// TIA Portal V17 export
// export: Created 2024-08-26T21:10:50.1762812Z, ExportSetting WithDefaults, DisplayName Totally Integrated Automation Portal, DisplayVersion V17 Update 7, DisplayName TIA Portal Openness, DisplayVersion V17 Update 7, DisplayName TIA Portal Version Control Interface, DisplayVersion V17, DisplayName SINAMICS Startdrive Advanced, DisplayVersion V17 SP2, DisplayName SINAMICS Startdrive G110M, G120, G120C, G120D, G120P, G115D, DisplayVersion V17 SP2, DisplayName SINAMICS Startdrive G130, G150, S120, S150, SINAMICS MV, S210, DisplayVersion V17 SP2, DisplayName STEP 7 Professional, DisplayVersion V17 Update 7, DisplayName STEP 7 Safety, DisplayVersion V17 Update 6, DisplayName WinCC Advanced / Unified PC, DisplayVersion V17 Update 7
FUNCTION "stationAlarms" : Void   // FC2, LAD
{ S7_Optimized_Access := 'TRUE' }
VERSION : 0.1
// stored: AutoNumber true, IsIECCheckEnabled false, SetENOAutomatically false, UDAEnableTagReadback false
   VAR_TEMP   // added for the SCL form of the ladder/FBD networks
      _w1 : Bool;
      _w2 : Bool;
      _w3 : Bool;
      _w4 : Bool;
      _w5 : Bool;
   END_VAR
BEGIN

REGION Network 1: ACTIVE ALARM
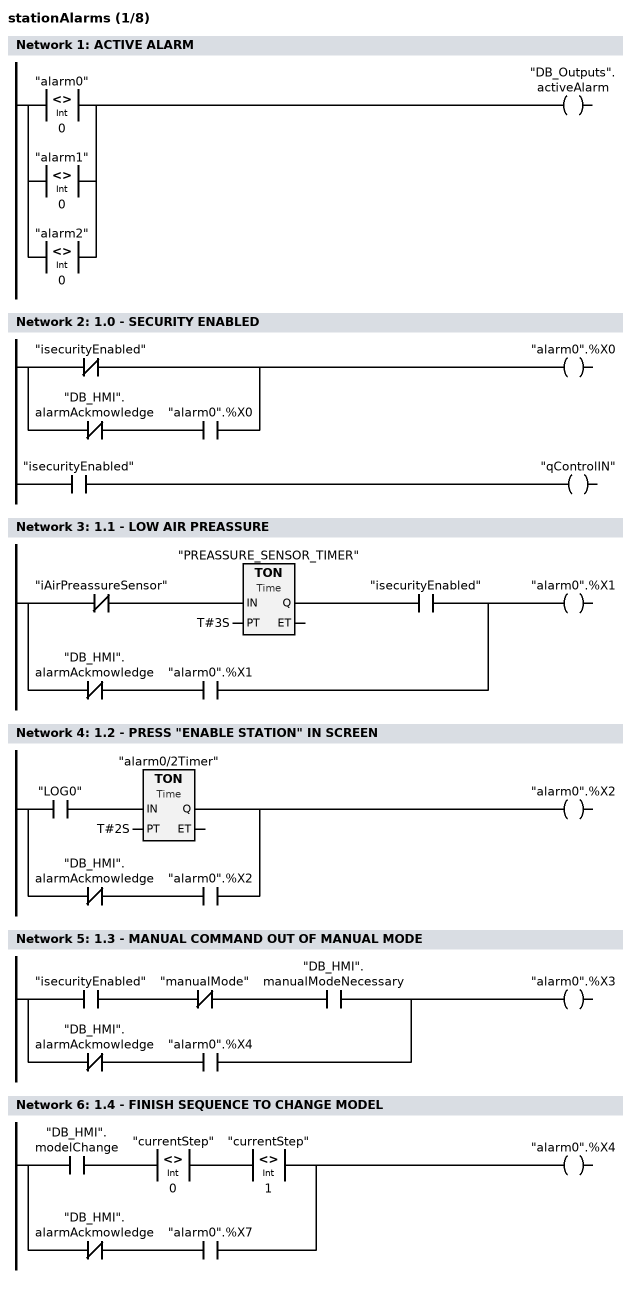
   RUNG wire#powerrail
      { S7_Templates := "SrcType := Int" } NE_Contact(in1 := "alarm0", in2 := 0)
      wire#w1
      Coil( "DB_Outputs".activeAlarm )
   END_RUNG
   RUNG wire#powerrail
      { S7_Templates := "SrcType := Int" } NE_Contact(in1 := "alarm1", in2 := 0)
   END_RUNG wire#w1
   RUNG wire#powerrail
      { S7_Templates := "SrcType := Int" } NE_Contact(in1 := "alarm2", in2 := 0)
   END_RUNG wire#w1
   // the same network as SCL:
   "DB_Outputs".activeAlarm := ("alarm0" <> 0) OR ("alarm1" <> 0) OR ("alarm2" <> 0);
END_REGION

REGION Network 2: 1.0 - SECURITY ENABLED
   RUNG wire#powerrail
      I_Contact( "isecurityEnabled" )
      wire#w1
      Coil( "alarm0".%X0 )
   END_RUNG
   RUNG wire#powerrail
      I_Contact( "DB_HMI".alarmAckmowledge )
      Contact( "alarm0".%X0 )
   END_RUNG wire#w1
   RUNG wire#powerrail
      Contact( "isecurityEnabled" )
      Coil( "qControlIN" )
   END_RUNG
   // the same network as SCL:
   "alarm0".%X0 := NOT "isecurityEnabled" OR (NOT "DB_HMI".alarmAckmowledge AND "alarm0".%X0);
   "qControlIN" := "isecurityEnabled";
END_REGION

REGION Network 3: 1.1 - LOW AIR PREASSURE
   RUNG wire#powerrail
      I_Contact( "iAirPreassureSensor" )
      { S7_Templates := "time_type := Time" } "PREASSURE_SENSOR_TIMER".TON(pt := T#3S, et =>)
      Contact( "isecurityEnabled" )
      wire#w1
      Coil( "alarm0".%X1 )
   END_RUNG
   RUNG wire#powerrail
      I_Contact( "DB_HMI".alarmAckmowledge )
      Contact( "alarm0".%X1 )
   END_RUNG wire#w1
   // the same network as SCL:
   "PREASSURE_SENSOR_TIMER".TON(IN := NOT "iAirPreassureSensor", PT := T#3S);
   "alarm0".%X1 := ("PREASSURE_SENSOR_TIMER".Q AND "isecurityEnabled") OR (NOT "DB_HMI".alarmAckmowledge AND "alarm0".%X1);
END_REGION

REGION Network 4: 1.2 - PRESS "ENABLE STATION" IN SCREEN
   RUNG wire#powerrail
      Contact( "LOG0" )
      { S7_Templates := "time_type := Time" } "alarm0/2Timer".TON(pt := T#2S, et =>)
      wire#w1
      Coil( "alarm0".%X2 )
   END_RUNG
   RUNG wire#powerrail
      I_Contact( "DB_HMI".alarmAckmowledge )
      Contact( "alarm0".%X2 )
   END_RUNG wire#w1
   // the same network as SCL:
   "alarm0/2Timer".TON(IN := "LOG0", PT := T#2S);
   "alarm0".%X2 := "alarm0/2Timer".Q OR (NOT "DB_HMI".alarmAckmowledge AND "alarm0".%X2);
END_REGION

REGION Network 5: 1.3 - MANUAL COMMAND OUT OF MANUAL MODE
   RUNG wire#powerrail
      Contact( "isecurityEnabled" )
      I_Contact( "manualMode" )
      Contact( "DB_HMI".manualModeNecessary )
      wire#w1
      Coil( "alarm0".%X3 )
   END_RUNG
   RUNG wire#powerrail
      I_Contact( "DB_HMI".alarmAckmowledge )
      Contact( "alarm0".%X4 )
   END_RUNG wire#w1
   // the same network as SCL:
   "alarm0".%X3 := ("isecurityEnabled" AND NOT "manualMode" AND "DB_HMI".manualModeNecessary) OR (NOT "DB_HMI".alarmAckmowledge AND "alarm0".%X4);
END_REGION

REGION Network 6: 1.4 - FINISH SEQUENCE TO CHANGE MODEL
   RUNG wire#powerrail
      Contact( "DB_HMI".modelChange )
      { S7_Templates := "SrcType := Int" } NE_Contact(in1 := "currentStep", in2 := 0)
      { S7_Templates := "SrcType := Int" } NE_Contact(in1 := "currentStep", in2 := 1)
      wire#w1
      Coil( "alarm0".%X4 )
   END_RUNG
   RUNG wire#powerrail
      I_Contact( "DB_HMI".alarmAckmowledge )
      Contact( "alarm0".%X7 )
   END_RUNG wire#w1
   // the same network as SCL:
   "alarm0".%X4 := ("DB_HMI".modelChange AND ("currentStep" <> 0) AND ("currentStep" <> 1)) OR (NOT "DB_HMI".alarmAckmowledge AND "alarm0".%X7);
END_REGION

REGION Network 7: 1.5 - WRONG LABEL
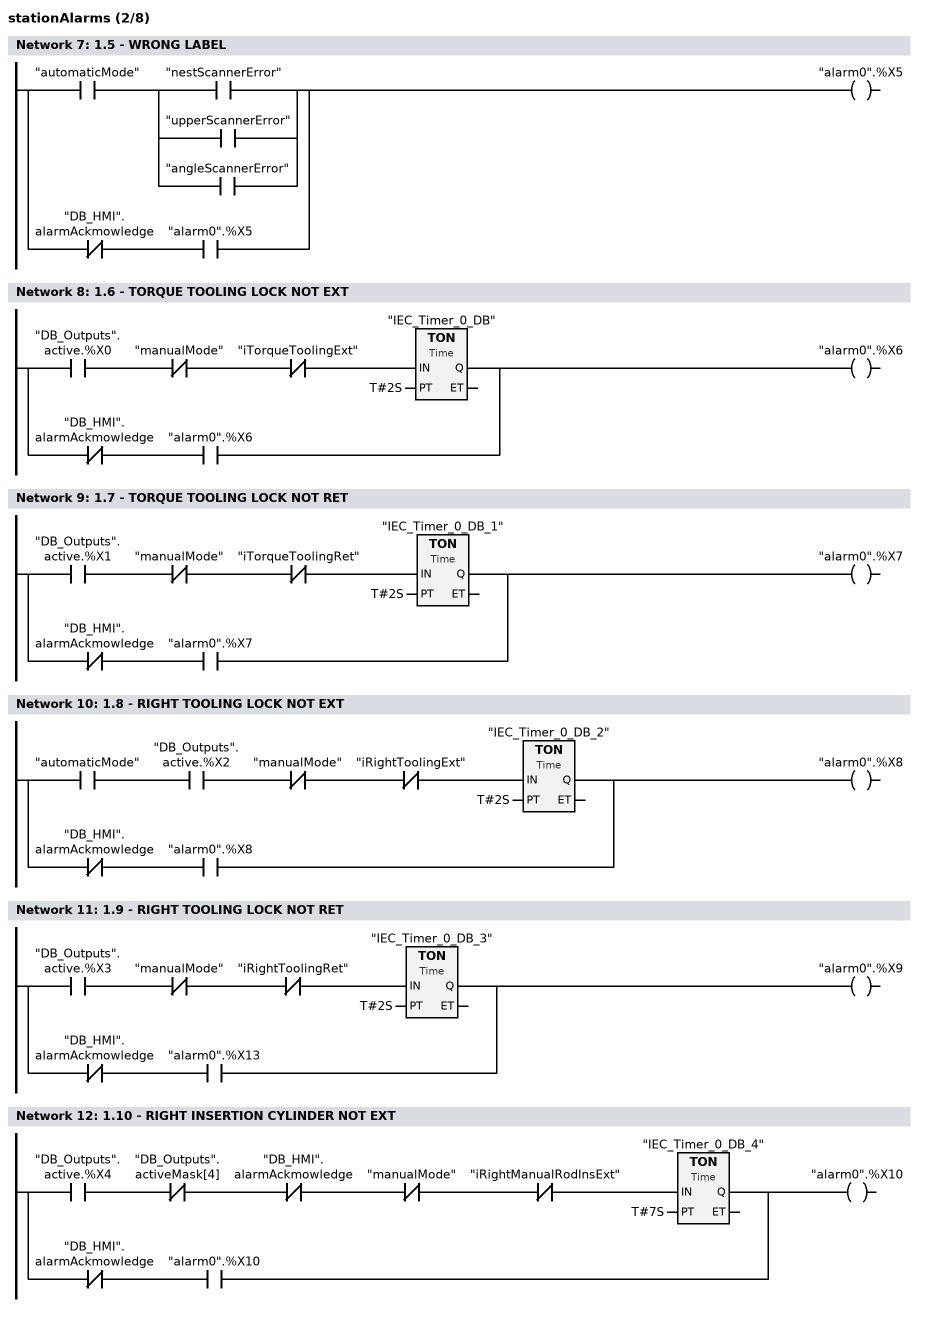
   RUNG wire#powerrail
      Contact( "automaticMode" )
      wire#w1
      Contact( "nestScannerError" )
      wire#w2
      Coil( "alarm0".%X5 )
   END_RUNG
   RUNG wire#w1
      Contact( "upperScannerError" )
   END_RUNG wire#w2
   RUNG wire#w1
      Contact( "angleScannerError" )
   END_RUNG wire#w2
   RUNG wire#powerrail
      I_Contact( "DB_HMI".alarmAckmowledge )
      Contact( "alarm0".%X5 )
   END_RUNG wire#w2
   // the same network as SCL:
   "alarm0".%X5 := ("automaticMode" AND ("nestScannerError" OR "upperScannerError" OR "angleScannerError")) OR (NOT "DB_HMI".alarmAckmowledge AND "alarm0".%X5);
END_REGION

REGION Network 8: 1.6 - TORQUE TOOLING LOCK NOT EXT
   RUNG wire#powerrail
      Contact( "DB_Outputs".active.%X0 )
      I_Contact( "manualMode" )
      I_Contact( "iTorqueToolingExt" )
      { S7_Templates := "time_type := Time" } "IEC_Timer_0_DB".TON(pt := T#2S, et =>)
      wire#w1
      Coil( "alarm0".%X6 )
   END_RUNG
   RUNG wire#powerrail
      I_Contact( "DB_HMI".alarmAckmowledge )
      Contact( "alarm0".%X6 )
   END_RUNG wire#w1
   // the same network as SCL:
   "IEC_Timer_0_DB".TON(IN := "DB_Outputs".active.%X0 AND NOT "manualMode" AND NOT "iTorqueToolingExt",
                        PT := T#2S);
   "alarm0".%X6 := "IEC_Timer_0_DB".Q OR (NOT "DB_HMI".alarmAckmowledge AND "alarm0".%X6);
END_REGION

REGION Network 9: 1.7 - TORQUE TOOLING LOCK NOT RET
   RUNG wire#powerrail
      Contact( "DB_Outputs".active.%X1 )
      I_Contact( "manualMode" )
      I_Contact( "iTorqueToolingRet" )
      { S7_Templates := "time_type := Time" } "IEC_Timer_0_DB_1".TON(pt := T#2S, et =>)
      wire#w1
      Coil( "alarm0".%X7 )
   END_RUNG
   RUNG wire#powerrail
      I_Contact( "DB_HMI".alarmAckmowledge )
      Contact( "alarm0".%X7 )
   END_RUNG wire#w1
   // the same network as SCL:
   "IEC_Timer_0_DB_1".TON(IN := "DB_Outputs".active.%X1 AND NOT "manualMode" AND NOT "iTorqueToolingRet",
                          PT := T#2S);
   "alarm0".%X7 := "IEC_Timer_0_DB_1".Q OR (NOT "DB_HMI".alarmAckmowledge AND "alarm0".%X7);
END_REGION

REGION Network 10: 1.8 - RIGHT TOOLING LOCK NOT EXT
   RUNG wire#powerrail
      Contact( "automaticMode" )
      Contact( "DB_Outputs".active.%X2 )
      I_Contact( "manualMode" )
      I_Contact( "iRightToolingExt" )
      { S7_Templates := "time_type := Time" } "IEC_Timer_0_DB_2".TON(pt := T#2S, et =>)
      wire#w1
      Coil( "alarm0".%X8 )
   END_RUNG
   RUNG wire#powerrail
      I_Contact( "DB_HMI".alarmAckmowledge )
      Contact( "alarm0".%X8 )
   END_RUNG wire#w1
   // the same network as SCL:
   "IEC_Timer_0_DB_2".TON(IN := "automaticMode" AND "DB_Outputs".active.%X2 AND NOT "manualMode" AND NOT "iRightToolingExt",
                          PT := T#2S);
   "alarm0".%X8 := "IEC_Timer_0_DB_2".Q OR (NOT "DB_HMI".alarmAckmowledge AND "alarm0".%X8);
END_REGION

REGION Network 11: 1.9 - RIGHT TOOLING LOCK NOT RET
   RUNG wire#powerrail
      Contact( "DB_Outputs".active.%X3 )
      I_Contact( "manualMode" )
      I_Contact( "iRightToolingRet" )
      { S7_Templates := "time_type := Time" } "IEC_Timer_0_DB_3".TON(pt := T#2S, et =>)
      wire#w1
      Coil( "alarm0".%X9 )
   END_RUNG
   RUNG wire#powerrail
      I_Contact( "DB_HMI".alarmAckmowledge )
      Contact( "alarm0".%X13 )
   END_RUNG wire#w1
   // the same network as SCL:
   "IEC_Timer_0_DB_3".TON(IN := "DB_Outputs".active.%X3 AND NOT "manualMode" AND NOT "iRightToolingRet",
                          PT := T#2S);
   "alarm0".%X9 := "IEC_Timer_0_DB_3".Q OR (NOT "DB_HMI".alarmAckmowledge AND "alarm0".%X13);
END_REGION

REGION Network 12: 1.10 - RIGHT INSERTION CYLINDER NOT EXT
   RUNG wire#powerrail
      Contact( "DB_Outputs".active.%X4 )
      I_Contact( "DB_Outputs".activeMask[4] )
      I_Contact( "DB_HMI".alarmAckmowledge )
      I_Contact( "manualMode" )
      I_Contact( "iRightManualRodInsExt" )
      { S7_Templates := "time_type := Time" } "IEC_Timer_0_DB_4".TON(pt := T#7S, et =>)
      wire#w1
      Coil( "alarm0".%X10 )
   END_RUNG
   RUNG wire#powerrail
      I_Contact( "DB_HMI".alarmAckmowledge )
      Contact( "alarm0".%X10 )
   END_RUNG wire#w1
   // the same network as SCL:
   "IEC_Timer_0_DB_4".TON(IN := "DB_Outputs".active.%X4 AND NOT "DB_Outputs".activeMask[4] AND NOT "DB_HMI".alarmAckmowledge AND NOT "manualMode" AND NOT "iRightManualRodInsExt",
                          PT := T#7S);
   "alarm0".%X10 := "IEC_Timer_0_DB_4".Q OR (NOT "DB_HMI".alarmAckmowledge AND "alarm0".%X10);
END_REGION

REGION Network 13: 1.11 - RIGHT INSERTION CYLINDER NOT RET
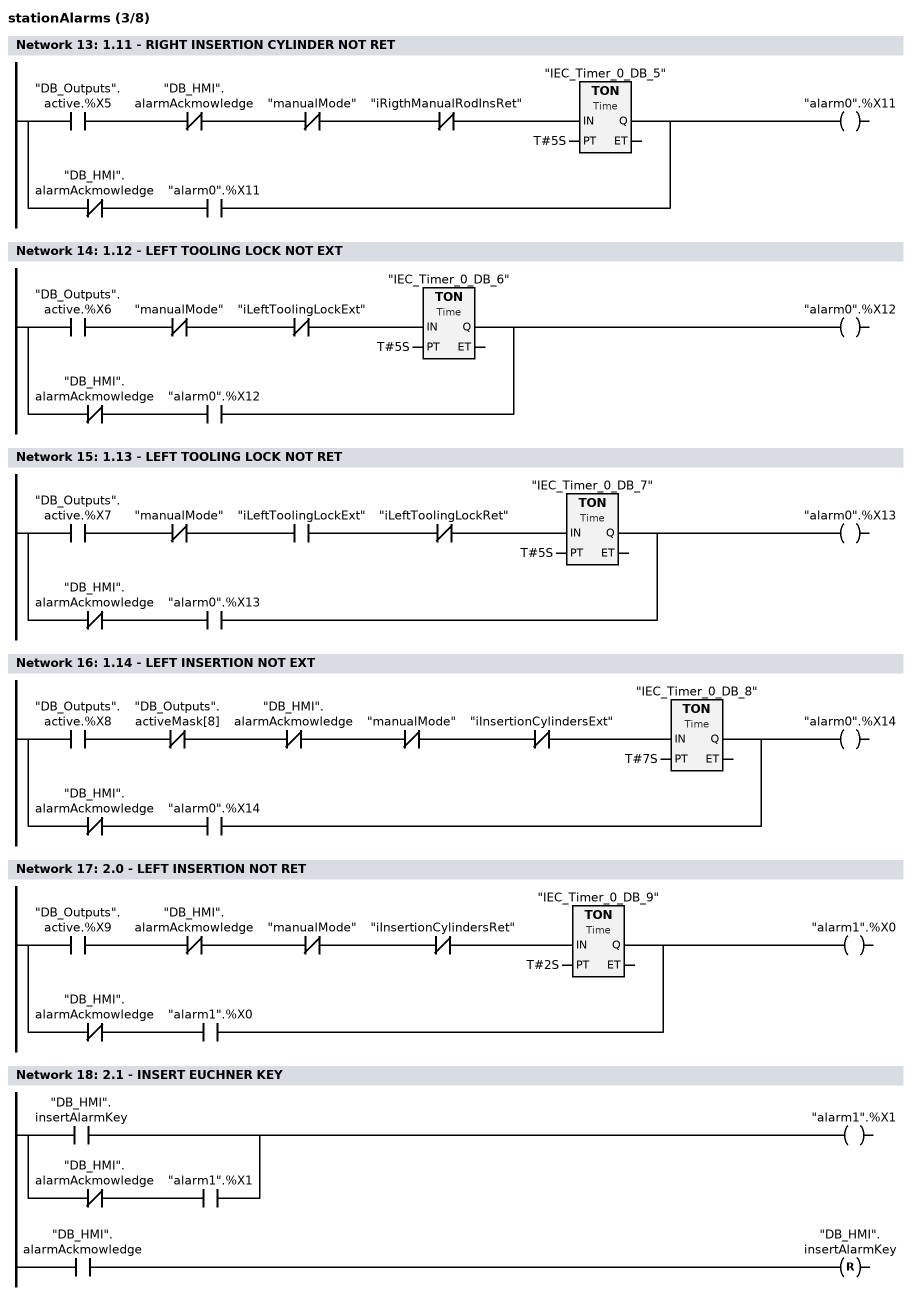
   RUNG wire#powerrail
      Contact( "DB_Outputs".active.%X5 )
      I_Contact( "DB_HMI".alarmAckmowledge )
      I_Contact( "manualMode" )
      I_Contact( "iRigthManualRodInsRet" )
      { S7_Templates := "time_type := Time" } "IEC_Timer_0_DB_5".TON(pt := T#5S, et =>)
      wire#w1
      Coil( "alarm0".%X11 )
   END_RUNG
   RUNG wire#powerrail
      I_Contact( "DB_HMI".alarmAckmowledge )
      Contact( "alarm0".%X11 )
   END_RUNG wire#w1
   // the same network as SCL:
   "IEC_Timer_0_DB_5".TON(IN := "DB_Outputs".active.%X5 AND NOT "DB_HMI".alarmAckmowledge AND NOT "manualMode" AND NOT "iRigthManualRodInsRet",
                          PT := T#5S);
   "alarm0".%X11 := "IEC_Timer_0_DB_5".Q OR (NOT "DB_HMI".alarmAckmowledge AND "alarm0".%X11);
END_REGION

REGION Network 14: 1.12 - LEFT TOOLING LOCK NOT EXT
   RUNG wire#powerrail
      Contact( "DB_Outputs".active.%X6 )
      I_Contact( "manualMode" )
      I_Contact( "iLeftToolingLockExt" )
      { S7_Templates := "time_type := Time" } "IEC_Timer_0_DB_6".TON(pt := T#5S, et =>)
      wire#w1
      Coil( "alarm0".%X12 )
   END_RUNG
   RUNG wire#powerrail
      I_Contact( "DB_HMI".alarmAckmowledge )
      Contact( "alarm0".%X12 )
   END_RUNG wire#w1
   // the same network as SCL:
   "IEC_Timer_0_DB_6".TON(IN := "DB_Outputs".active.%X6 AND NOT "manualMode" AND NOT "iLeftToolingLockExt",
                          PT := T#5S);
   "alarm0".%X12 := "IEC_Timer_0_DB_6".Q OR (NOT "DB_HMI".alarmAckmowledge AND "alarm0".%X12);
END_REGION

REGION Network 15: 1.13 - LEFT TOOLING LOCK NOT RET
   RUNG wire#powerrail
      Contact( "DB_Outputs".active.%X7 )
      I_Contact( "manualMode" )
      Contact( "iLeftToolingLockExt" )
      I_Contact( "iLeftToolingLockRet" )
      { S7_Templates := "time_type := Time" } "IEC_Timer_0_DB_7".TON(pt := T#5S, et =>)
      wire#w1
      Coil( "alarm0".%X13 )
   END_RUNG
   RUNG wire#powerrail
      I_Contact( "DB_HMI".alarmAckmowledge )
      Contact( "alarm0".%X13 )
   END_RUNG wire#w1
   // the same network as SCL:
   "IEC_Timer_0_DB_7".TON(IN := "DB_Outputs".active.%X7 AND NOT "manualMode" AND "iLeftToolingLockExt" AND NOT "iLeftToolingLockRet",
                          PT := T#5S);
   "alarm0".%X13 := "IEC_Timer_0_DB_7".Q OR (NOT "DB_HMI".alarmAckmowledge AND "alarm0".%X13);
END_REGION

REGION Network 16: 1.14 - LEFT INSERTION NOT EXT
   RUNG wire#powerrail
      Contact( "DB_Outputs".active.%X8 )
      I_Contact( "DB_Outputs".activeMask[8] )
      I_Contact( "DB_HMI".alarmAckmowledge )
      I_Contact( "manualMode" )
      I_Contact( "iInsertionCylindersExt" )
      { S7_Templates := "time_type := Time" } "IEC_Timer_0_DB_8".TON(pt := T#7S, et =>)
      wire#w1
      Coil( "alarm0".%X14 )
   END_RUNG
   RUNG wire#powerrail
      I_Contact( "DB_HMI".alarmAckmowledge )
      Contact( "alarm0".%X14 )
   END_RUNG wire#w1
   // the same network as SCL:
   "IEC_Timer_0_DB_8".TON(IN := "DB_Outputs".active.%X8 AND NOT "DB_Outputs".activeMask[8] AND NOT "DB_HMI".alarmAckmowledge AND NOT "manualMode" AND NOT "iInsertionCylindersExt",
                          PT := T#7S);
   "alarm0".%X14 := "IEC_Timer_0_DB_8".Q OR (NOT "DB_HMI".alarmAckmowledge AND "alarm0".%X14);
END_REGION

REGION Network 17: 2.0 - LEFT INSERTION NOT RET
   RUNG wire#powerrail
      Contact( "DB_Outputs".active.%X9 )
      I_Contact( "DB_HMI".alarmAckmowledge )
      I_Contact( "manualMode" )
      I_Contact( "iInsertionCylindersRet" )
      { S7_Templates := "time_type := Time" } "IEC_Timer_0_DB_9".TON(pt := T#2S, et =>)
      wire#w1
      Coil( "alarm1".%X0 )
   END_RUNG
   RUNG wire#powerrail
      I_Contact( "DB_HMI".alarmAckmowledge )
      Contact( "alarm1".%X0 )
   END_RUNG wire#w1
   // the same network as SCL:
   "IEC_Timer_0_DB_9".TON(IN := "DB_Outputs".active.%X9 AND NOT "DB_HMI".alarmAckmowledge AND NOT "manualMode" AND NOT "iInsertionCylindersRet",
                          PT := T#2S);
   "alarm1".%X0 := "IEC_Timer_0_DB_9".Q OR (NOT "DB_HMI".alarmAckmowledge AND "alarm1".%X0);
END_REGION

REGION Network 18: 2.1 - INSERT EUCHNER KEY
   RUNG wire#powerrail
      Contact( "DB_HMI".insertAlarmKey )
      wire#w1
      Coil( "alarm1".%X1 )
   END_RUNG
   RUNG wire#powerrail
      I_Contact( "DB_HMI".alarmAckmowledge )
      Contact( "alarm1".%X1 )
   END_RUNG wire#w1
   RUNG wire#powerrail
      Contact( "DB_HMI".alarmAckmowledge )
      R_Coil( "DB_HMI".insertAlarmKey )
   END_RUNG
   // the same network as SCL:
   "alarm1".%X1 := "DB_HMI".insertAlarmKey OR (NOT "DB_HMI".alarmAckmowledge AND "alarm1".%X1);
   IF "DB_HMI".alarmAckmowledge THEN "DB_HMI".insertAlarmKey := FALSE; END_IF;
END_REGION

REGION Network 19: 2.2 - TORQUE NOK RESTART
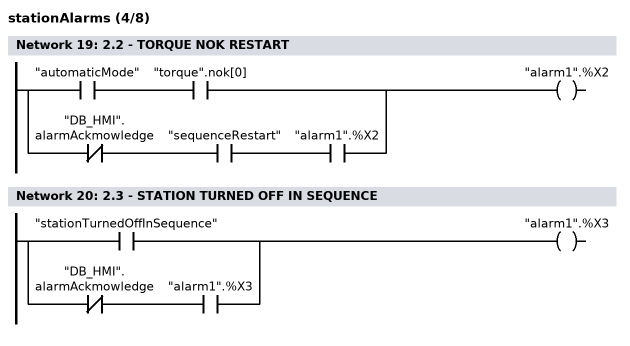
   RUNG wire#powerrail
      Contact( "automaticMode" )
      Contact( "torque".nok[0] )
      wire#w1
      Coil( "alarm1".%X2 )
   END_RUNG
   RUNG wire#powerrail
      I_Contact( "DB_HMI".alarmAckmowledge )
      Contact( "sequenceRestart" )
      Contact( "alarm1".%X2 )
   END_RUNG wire#w1
   // the same network as SCL:
   "alarm1".%X2 := ("automaticMode" AND "torque".nok[0]) OR (NOT "DB_HMI".alarmAckmowledge AND "sequenceRestart" AND "alarm1".%X2);
END_REGION

REGION Network 20: 2.3 - STATION TURNED OFF IN SEQUENCE
   RUNG wire#powerrail
      Contact( "stationTurnedOffInSequence" )
      wire#w1
      Coil( "alarm1".%X3 )
   END_RUNG
   RUNG wire#powerrail
      I_Contact( "DB_HMI".alarmAckmowledge )
      Contact( "alarm1".%X3 )
   END_RUNG wire#w1
   // the same network as SCL:
   "alarm1".%X3 := "stationTurnedOffInSequence" OR (NOT "DB_HMI".alarmAckmowledge AND "alarm1".%X3);
END_REGION

REGION Network 21: 2.4-2.13 - COMMUNICATION ALARMS
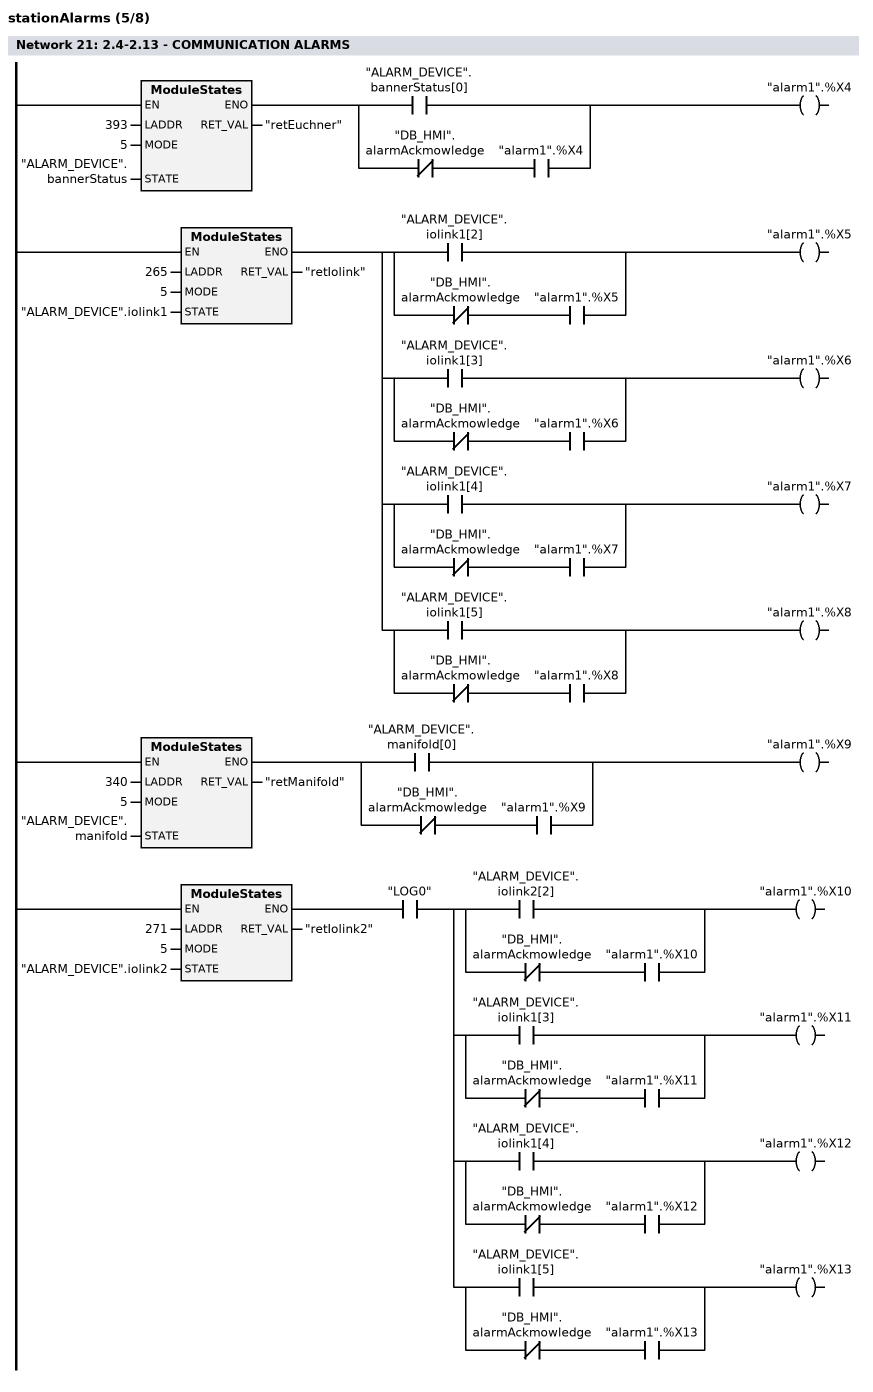
   RUNG wire#powerrail
      ModuleStates(LADDR := 393, MODE := 5, STATE := "ALARM_DEVICE".bannerStatus, Ret_Val => "retEuchner")
      wire#w1
      Contact( "ALARM_DEVICE".bannerStatus[0] )
      wire#w2
      Coil( "alarm1".%X4 )
   END_RUNG
   RUNG wire#w1
      I_Contact( "DB_HMI".alarmAckmowledge )
      Contact( "alarm1".%X4 )
   END_RUNG wire#w2
   RUNG wire#powerrail
      ModuleStates(LADDR := 265, MODE := 5, STATE := "ALARM_DEVICE".iolink1, Ret_Val => "retIolink")
      wire#w3
      Contact( "ALARM_DEVICE".iolink1[2] )
      wire#w4
      Coil( "alarm1".%X5 )
   END_RUNG
   RUNG wire#w3
      I_Contact( "DB_HMI".alarmAckmowledge )
      Contact( "alarm1".%X5 )
   END_RUNG wire#w4
   RUNG wire#w3
      Contact( "ALARM_DEVICE".iolink1[3] )
      wire#w5
      Coil( "alarm1".%X6 )
   END_RUNG
   RUNG wire#w3
      I_Contact( "DB_HMI".alarmAckmowledge )
      Contact( "alarm1".%X6 )
   END_RUNG wire#w5
   RUNG wire#w3
      Contact( "ALARM_DEVICE".iolink1[4] )
      wire#w6
      Coil( "alarm1".%X7 )
   END_RUNG
   RUNG wire#w3
      I_Contact( "DB_HMI".alarmAckmowledge )
      Contact( "alarm1".%X7 )
   END_RUNG wire#w6
   RUNG wire#w3
      Contact( "ALARM_DEVICE".iolink1[5] )
      wire#w7
      Coil( "alarm1".%X8 )
   END_RUNG
   RUNG wire#w3
      I_Contact( "DB_HMI".alarmAckmowledge )
      Contact( "alarm1".%X8 )
   END_RUNG wire#w7
   RUNG wire#powerrail
      ModuleStates(LADDR := 340, MODE := 5, STATE := "ALARM_DEVICE".manifold, Ret_Val => "retManifold")
      wire#w8
      Contact( "ALARM_DEVICE".manifold[0] )
      wire#w9
      Coil( "alarm1".%X9 )
   END_RUNG
   RUNG wire#w8
      I_Contact( "DB_HMI".alarmAckmowledge )
      Contact( "alarm1".%X9 )
   END_RUNG wire#w9
   RUNG wire#powerrail
      ModuleStates(LADDR := 271, MODE := 5, STATE := "ALARM_DEVICE".iolink2, Ret_Val => "retIolink2")
      Contact( "LOG0" )
      wire#w10
      Contact( "ALARM_DEVICE".iolink2[2] )
      wire#w11
      Coil( "alarm1".%X10 )
   END_RUNG
   RUNG wire#w10
      I_Contact( "DB_HMI".alarmAckmowledge )
      Contact( "alarm1".%X10 )
   END_RUNG wire#w11
   RUNG wire#w10
      Contact( "ALARM_DEVICE".iolink1[3] )
      wire#w12
      Coil( "alarm1".%X11 )
   END_RUNG
   RUNG wire#w10
      I_Contact( "DB_HMI".alarmAckmowledge )
      Contact( "alarm1".%X11 )
   END_RUNG wire#w12
   RUNG wire#w10
      Contact( "ALARM_DEVICE".iolink1[4] )
      wire#w13
      Coil( "alarm1".%X12 )
   END_RUNG
   RUNG wire#w10
      I_Contact( "DB_HMI".alarmAckmowledge )
      Contact( "alarm1".%X12 )
   END_RUNG wire#w13
   RUNG wire#w10
      Contact( "ALARM_DEVICE".iolink1[5] )
      wire#w14
      Coil( "alarm1".%X13 )
   END_RUNG
   RUNG wire#w10
      I_Contact( "DB_HMI".alarmAckmowledge )
      Contact( "alarm1".%X13 )
   END_RUNG wire#w14
   // the same network as SCL:
   "retEuchner" := ModuleStates(LADDR := 393, MODE := 5, STATE := "ALARM_DEVICE".bannerStatus, ENO => #_w1);
   "alarm1".%X4 := #_w1 AND ("ALARM_DEVICE".bannerStatus[0] OR (NOT "DB_HMI".alarmAckmowledge AND "alarm1".%X4));
   "retIolink" := ModuleStates(LADDR := 265, MODE := 5, STATE := "ALARM_DEVICE".iolink1, ENO => #_w2);
   "alarm1".%X5 := #_w2 AND ("ALARM_DEVICE".iolink1[2] OR (NOT "DB_HMI".alarmAckmowledge AND "alarm1".%X5));
   "alarm1".%X6 := #_w2 AND ("ALARM_DEVICE".iolink1[3] OR (NOT "DB_HMI".alarmAckmowledge AND "alarm1".%X6));
   "alarm1".%X7 := #_w2 AND ("ALARM_DEVICE".iolink1[4] OR (NOT "DB_HMI".alarmAckmowledge AND "alarm1".%X7));
   "alarm1".%X8 := #_w2 AND ("ALARM_DEVICE".iolink1[5] OR (NOT "DB_HMI".alarmAckmowledge AND "alarm1".%X8));
   "retManifold" := ModuleStates(LADDR := 340, MODE := 5, STATE := "ALARM_DEVICE".manifold, ENO => #_w3);
   "alarm1".%X9 := #_w3 AND ("ALARM_DEVICE".manifold[0] OR (NOT "DB_HMI".alarmAckmowledge AND "alarm1".%X9));
   "retIolink2" := ModuleStates(LADDR := 271, MODE := 5, STATE := "ALARM_DEVICE".iolink2, ENO => #_w4);
   #_w5 := #_w4 AND "LOG0";
   "alarm1".%X10 := #_w5 AND ("ALARM_DEVICE".iolink2[2] OR (NOT "DB_HMI".alarmAckmowledge AND "alarm1".%X10));
   "alarm1".%X11 := #_w5 AND ("ALARM_DEVICE".iolink1[3] OR (NOT "DB_HMI".alarmAckmowledge AND "alarm1".%X11));
   "alarm1".%X12 := #_w5 AND ("ALARM_DEVICE".iolink1[4] OR (NOT "DB_HMI".alarmAckmowledge AND "alarm1".%X12));
   "alarm1".%X13 := #_w5 AND ("ALARM_DEVICE".iolink1[5] OR (NOT "DB_HMI".alarmAckmowledge AND "alarm1".%X13));
END_REGION

REGION Network 22: 2.14.- TORQUE TO ACTIVATION POS
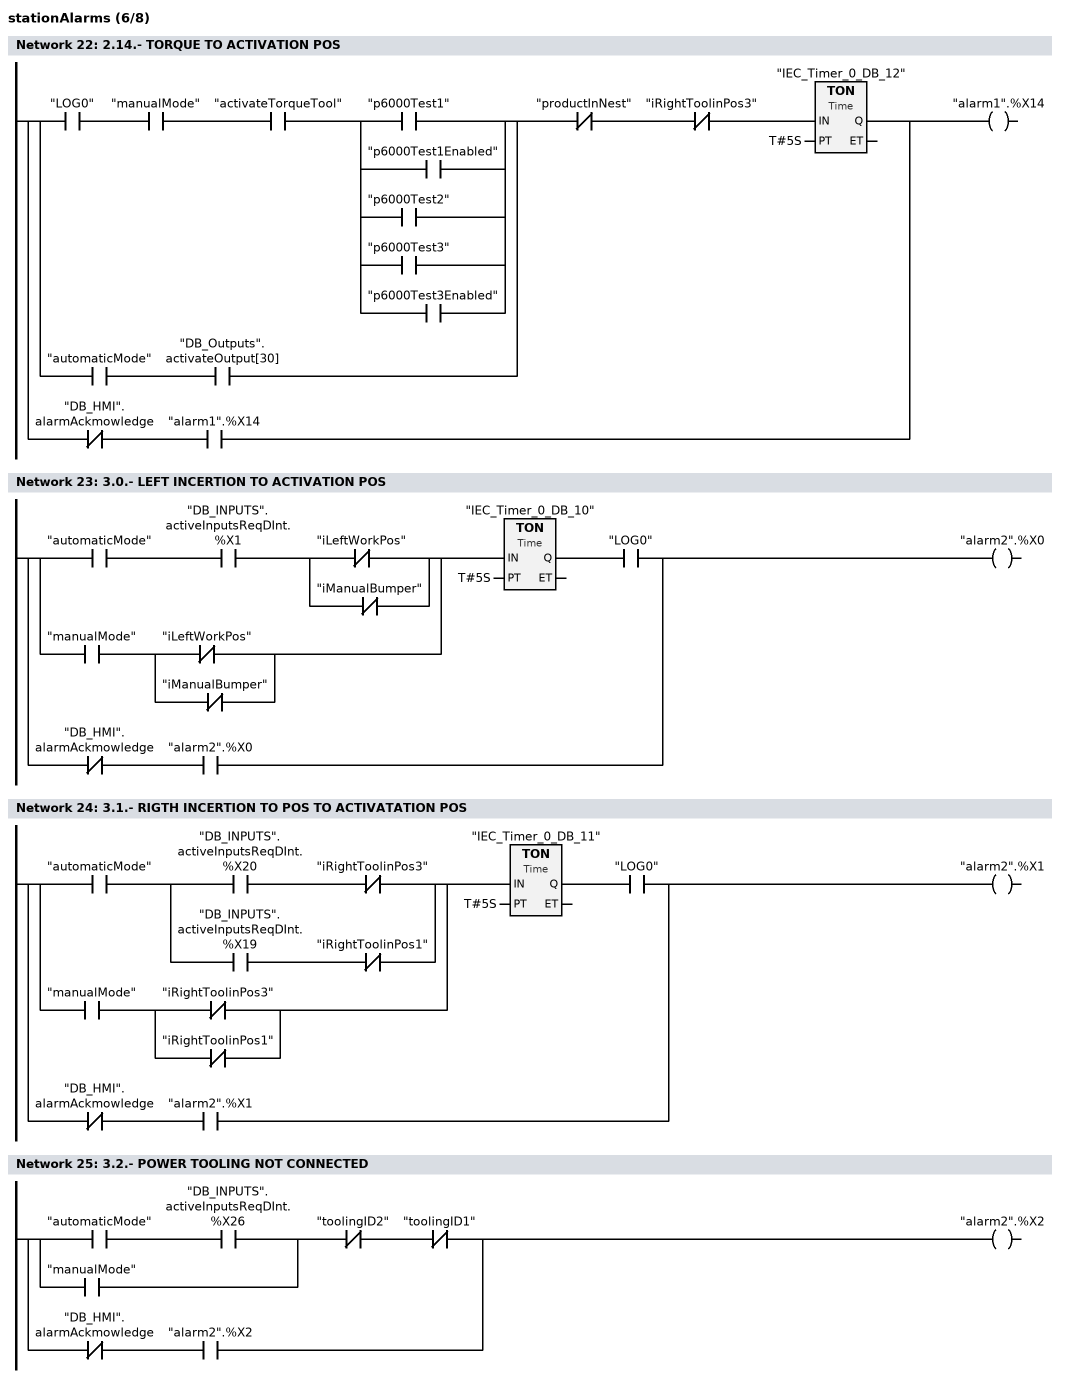
   RUNG wire#powerrail
      Contact( "LOG0" )
      Contact( "manualMode" )
      Contact( "activateTorqueTool" )
      wire#w1
      Contact( "p6000Test1" )
      wire#w2
      I_Contact( "productInNest" )
      I_Contact( "iRightToolinPos3" )
      { S7_Templates := "time_type := Time" } "IEC_Timer_0_DB_12".TON(pt := T#5S, et =>)
      wire#w3
      Coil( "alarm1".%X14 )
   END_RUNG
   RUNG wire#w1
      Contact( "p6000Test1Enabled" )
   END_RUNG wire#w2
   RUNG wire#w1
      Contact( "p6000Test2" )
   END_RUNG wire#w2
   RUNG wire#w1
      Contact( "p6000Test3" )
   END_RUNG wire#w2
   RUNG wire#w1
      Contact( "p6000Test3Enabled" )
   END_RUNG wire#w2
   RUNG wire#powerrail
      Contact( "automaticMode" )
      Contact( "DB_Outputs".activateOutput[30] )
   END_RUNG wire#w2
   RUNG wire#powerrail
      I_Contact( "DB_HMI".alarmAckmowledge )
      Contact( "alarm1".%X14 )
   END_RUNG wire#w3
   // the same network as SCL:
   "IEC_Timer_0_DB_12".TON(IN := (("LOG0" AND "manualMode" AND "activateTorqueTool" AND ("p6000Test1" OR "p6000Test1Enabled" OR "p6000Test2" OR "p6000Test3" OR "p6000Test3Enabled")) OR ("automaticMode" AND "DB_Outputs".activateOutput[30])) AND NOT "productInNest" AND NOT "iRightToolinPos3",
                           PT := T#5S);
   "alarm1".%X14 := "IEC_Timer_0_DB_12".Q OR (NOT "DB_HMI".alarmAckmowledge AND "alarm1".%X14);
END_REGION

REGION Network 23: 3.0.- LEFT INCERTION TO ACTIVATION POS
   RUNG wire#powerrail
      Contact( "automaticMode" )
      Contact( "DB_INPUTS".activeInputsReqDInt.%X1 )
      wire#w1
      I_Contact( "iLeftWorkPos" )
      wire#w2
      { S7_Templates := "time_type := Time" } "IEC_Timer_0_DB_10".TON(pt := T#5S, et =>)
      Contact( "LOG0" )
      wire#w4
      Coil( "alarm2".%X0 )
   END_RUNG
   RUNG wire#w1
      I_Contact( "iManualBumper" )
   END_RUNG wire#w2
   RUNG wire#powerrail
      Contact( "manualMode" )
      wire#w3
      I_Contact( "iLeftWorkPos" )
   END_RUNG wire#w2
   RUNG wire#w3
      I_Contact( "iManualBumper" )
   END_RUNG wire#w2
   RUNG wire#powerrail
      I_Contact( "DB_HMI".alarmAckmowledge )
      Contact( "alarm2".%X0 )
   END_RUNG wire#w4
   // the same network as SCL:
   "IEC_Timer_0_DB_10".TON(IN := ("automaticMode" AND "DB_INPUTS".activeInputsReqDInt.%X1 AND (NOT "iLeftWorkPos" OR NOT "iManualBumper")) OR ("manualMode" AND (NOT "iLeftWorkPos" OR NOT "iManualBumper")),
                           PT := T#5S);
   "alarm2".%X0 := ("IEC_Timer_0_DB_10".Q AND "LOG0") OR (NOT "DB_HMI".alarmAckmowledge AND "alarm2".%X0);
END_REGION

REGION Network 24: 3.1.- RIGTH INCERTION TO POS TO ACTIVATATION POS
   RUNG wire#powerrail
      Contact( "automaticMode" )
      wire#w1
      Contact( "DB_INPUTS".activeInputsReqDInt.%X20 )
      I_Contact( "iRightToolinPos3" )
      wire#w2
      { S7_Templates := "time_type := Time" } "IEC_Timer_0_DB_11".TON(pt := T#5S, et =>)
      Contact( "LOG0" )
      wire#w4
      Coil( "alarm2".%X1 )
   END_RUNG
   RUNG wire#w1
      Contact( "DB_INPUTS".activeInputsReqDInt.%X19 )
      I_Contact( "iRightToolinPos1" )
   END_RUNG wire#w2
   RUNG wire#powerrail
      Contact( "manualMode" )
      wire#w3
      I_Contact( "iRightToolinPos3" )
   END_RUNG wire#w2
   RUNG wire#w3
      I_Contact( "iRightToolinPos1" )
   END_RUNG wire#w2
   RUNG wire#powerrail
      I_Contact( "DB_HMI".alarmAckmowledge )
      Contact( "alarm2".%X1 )
   END_RUNG wire#w4
   // the same network as SCL:
   "IEC_Timer_0_DB_11".TON(IN := ("automaticMode" AND (("DB_INPUTS".activeInputsReqDInt.%X20 AND NOT "iRightToolinPos3") OR ("DB_INPUTS".activeInputsReqDInt.%X19 AND NOT "iRightToolinPos1"))) OR ("manualMode" AND (NOT "iRightToolinPos3" OR NOT "iRightToolinPos1")),
                           PT := T#5S);
   "alarm2".%X1 := ("IEC_Timer_0_DB_11".Q AND "LOG0") OR (NOT "DB_HMI".alarmAckmowledge AND "alarm2".%X1);
END_REGION

REGION Network 25: 3.2.- POWER TOOLING NOT CONNECTED
   RUNG wire#powerrail
      Contact( "automaticMode" )
      Contact( "DB_INPUTS".activeInputsReqDInt.%X26 )
      wire#w1
      I_Contact( "toolingID2" )
      I_Contact( "toolingID1" )
      wire#w2
      Coil( "alarm2".%X2 )
   END_RUNG
   RUNG wire#powerrail
      Contact( "manualMode" )
   END_RUNG wire#w1
   RUNG wire#powerrail
      I_Contact( "DB_HMI".alarmAckmowledge )
      Contact( "alarm2".%X2 )
   END_RUNG wire#w2
   // the same network as SCL:
   "alarm2".%X2 := ((("automaticMode" AND "DB_INPUTS".activeInputsReqDInt.%X26) OR "manualMode") AND NOT "toolingID2" AND NOT "toolingID1") OR (NOT "DB_HMI".alarmAckmowledge AND "alarm2".%X2);
END_REGION

REGION Network 26: 3.3.- MANUAL TOOLING NOT CONNECTED
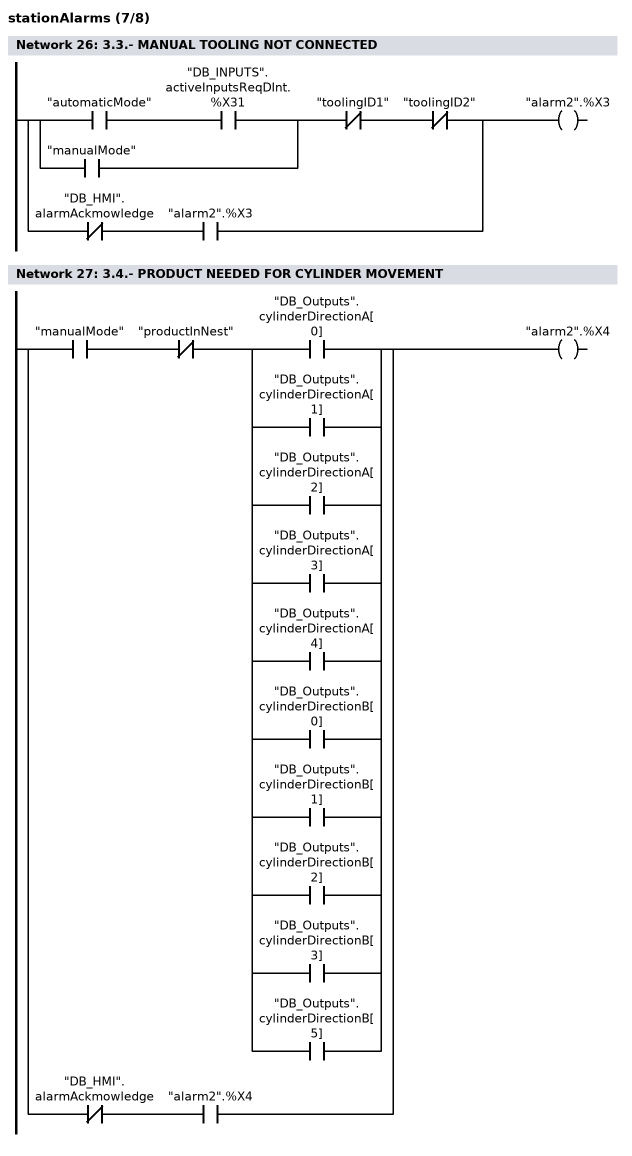
   RUNG wire#powerrail
      Contact( "automaticMode" )
      Contact( "DB_INPUTS".activeInputsReqDInt.%X31 )
      wire#w1
      I_Contact( "toolingID1" )
      I_Contact( "toolingID2" )
      wire#w2
      Coil( "alarm2".%X3 )
   END_RUNG
   RUNG wire#powerrail
      Contact( "manualMode" )
   END_RUNG wire#w1
   RUNG wire#powerrail
      I_Contact( "DB_HMI".alarmAckmowledge )
      Contact( "alarm2".%X3 )
   END_RUNG wire#w2
   // the same network as SCL:
   "alarm2".%X3 := ((("automaticMode" AND "DB_INPUTS".activeInputsReqDInt.%X31) OR "manualMode") AND NOT "toolingID1" AND NOT "toolingID2") OR (NOT "DB_HMI".alarmAckmowledge AND "alarm2".%X3);
END_REGION

REGION Network 27: 3.4.- PRODUCT NEEDED FOR CYLINDER MOVEMENT
   RUNG wire#powerrail
      Contact( "manualMode" )
      I_Contact( "productInNest" )
      wire#w1
      Contact( "DB_Outputs".cylinderDirectionA[0] )
      wire#w2
      Coil( "alarm2".%X4 )
   END_RUNG
   RUNG wire#w1
      Contact( "DB_Outputs".cylinderDirectionA[1] )
   END_RUNG wire#w2
   RUNG wire#w1
      Contact( "DB_Outputs".cylinderDirectionA[2] )
   END_RUNG wire#w2
   RUNG wire#w1
      Contact( "DB_Outputs".cylinderDirectionA[3] )
   END_RUNG wire#w2
   RUNG wire#w1
      Contact( "DB_Outputs".cylinderDirectionA[4] )
   END_RUNG wire#w2
   RUNG wire#w1
      Contact( "DB_Outputs".cylinderDirectionB[0] )
   END_RUNG wire#w2
   RUNG wire#w1
      Contact( "DB_Outputs".cylinderDirectionB[1] )
   END_RUNG wire#w2
   RUNG wire#w1
      Contact( "DB_Outputs".cylinderDirectionB[2] )
   END_RUNG wire#w2
   RUNG wire#w1
      Contact( "DB_Outputs".cylinderDirectionB[3] )
   END_RUNG wire#w2
   RUNG wire#w1
      Contact( "DB_Outputs".cylinderDirectionB[5] )
   END_RUNG wire#w2
   RUNG wire#powerrail
      I_Contact( "DB_HMI".alarmAckmowledge )
      Contact( "alarm2".%X4 )
   END_RUNG wire#w2
   // the same network as SCL:
   "alarm2".%X4 := ("manualMode" AND NOT "productInNest" AND ("DB_Outputs".cylinderDirectionA[0] OR "DB_Outputs".cylinderDirectionA[1] OR "DB_Outputs".cylinderDirectionA[2] OR "DB_Outputs".cylinderDirectionA[3] OR "DB_Outputs".cylinderDirectionA[4] OR "DB_Outputs".cylinderDirectionB[0] OR "DB_Outputs".cylinderDirectionB[1] OR "DB_Outputs".cylinderDirectionB[2] OR "DB_Outputs".cylinderDirectionB[3] OR "DB_Outputs".cylinderDirectionB[5])) OR (NOT "DB_HMI".alarmAckmowledge AND "alarm2".%X4);
END_REGION

REGION Network 28: 3.5.- MAN LH PROD NOK ROD
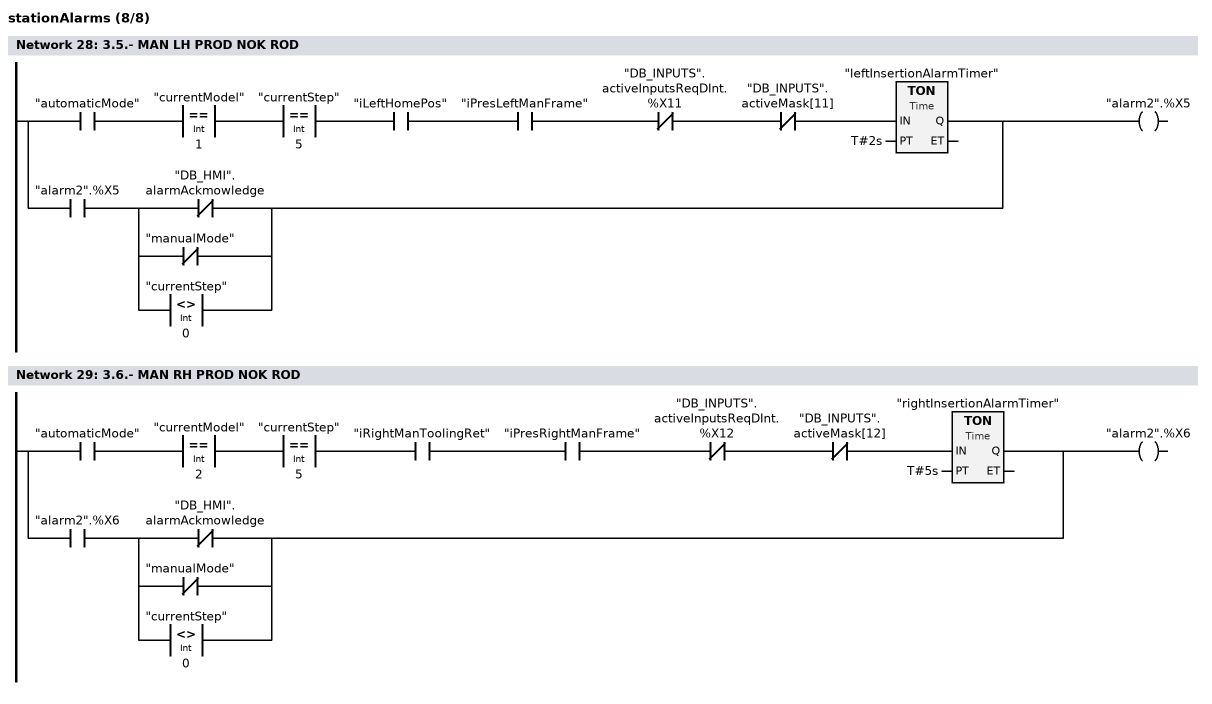
   RUNG wire#powerrail
      Contact( "automaticMode" )
      { S7_Templates := "SrcType := Int" } EQ_Contact(in1 := "currentModel", in2 := 1)
      { S7_Templates := "SrcType := Int" } EQ_Contact(in1 := "currentStep", in2 := 5)
      Contact( "iLeftHomePos" )
      Contact( "iPresLeftManFrame" )
      I_Contact( "DB_INPUTS".activeInputsReqDInt.%X11 )
      I_Contact( "DB_INPUTS".activeMask[11] )
      { S7_Templates := "time_type := Time" } "leftInsertionAlarmTimer".TON(pt := T#2s, et =>)
      wire#w1
      Coil( "alarm2".%X5 )
   END_RUNG
   RUNG wire#powerrail
      Contact( "alarm2".%X5 )
      wire#w2
      I_Contact( "DB_HMI".alarmAckmowledge )
   END_RUNG wire#w1
   RUNG wire#w2
      I_Contact( "manualMode" )
   END_RUNG wire#w1
   RUNG wire#w2
      { S7_Templates := "SrcType := Int" } NE_Contact(in1 := "currentStep", in2 := 0)
   END_RUNG wire#w1
   // the same network as SCL:
   "leftInsertionAlarmTimer".TON(IN := "automaticMode" AND ("currentModel" = 1) AND ("currentStep" = 5) AND "iLeftHomePos" AND "iPresLeftManFrame" AND NOT "DB_INPUTS".activeInputsReqDInt.%X11 AND NOT "DB_INPUTS".activeMask[11],
                           PT := T#2s);
   "alarm2".%X5 := "leftInsertionAlarmTimer".Q OR ("alarm2".%X5 AND (NOT "DB_HMI".alarmAckmowledge OR NOT "manualMode" OR ("currentStep" <> 0)));
END_REGION

REGION Network 29: 3.6.- MAN RH PROD NOK ROD
   RUNG wire#powerrail
      Contact( "automaticMode" )
      { S7_Templates := "SrcType := Int" } EQ_Contact(in1 := "currentModel", in2 := 2)
      { S7_Templates := "SrcType := Int" } EQ_Contact(in1 := "currentStep", in2 := 5)
      Contact( "iRightManToolingRet" )
      Contact( "iPresRightManFrame" )
      I_Contact( "DB_INPUTS".activeInputsReqDInt.%X12 )
      I_Contact( "DB_INPUTS".activeMask[12] )
      { S7_Templates := "time_type := Time" } "rightInsertionAlarmTimer".TON(pt := T#5s, et =>)
      wire#w1
      Coil( "alarm2".%X6 )
   END_RUNG
   RUNG wire#powerrail
      Contact( "alarm2".%X6 )
      wire#w2
      I_Contact( "DB_HMI".alarmAckmowledge )
   END_RUNG wire#w1
   RUNG wire#w2
      I_Contact( "manualMode" )
   END_RUNG wire#w1
   RUNG wire#w2
      { S7_Templates := "SrcType := Int" } NE_Contact(in1 := "currentStep", in2 := 0)
   END_RUNG wire#w1
   // the same network as SCL:
   "rightInsertionAlarmTimer".TON(IN := "automaticMode" AND ("currentModel" = 2) AND ("currentStep" = 5) AND "iRightManToolingRet" AND "iPresRightManFrame" AND NOT "DB_INPUTS".activeInputsReqDInt.%X12 AND NOT "DB_INPUTS".activeMask[12],
                           PT := T#5s);
   "alarm2".%X6 := "rightInsertionAlarmTimer".Q OR ("alarm2".%X6 AND (NOT "DB_HMI".alarmAckmowledge OR NOT "manualMode" OR ("currentStep" <> 0)));
END_REGION
END_FUNCTION
